FUNCTION_BLOCK Test_F_Equals EXTENDS TUnitTestBase
VAR
END_VAR

Assertion.AssertEquals_BOOL(
    Expected:= TRUE, 
    Actual:= F_Equals(1.000_005,1.000_004,0.000_002), 
    VariableName:= 'F_Equals');
    
Assertion.AssertEquals_BOOL(
    Expected:= FALSE, 
    Actual:= F_Equals(1.000_005,1.000_003,0.000_001), 
    VariableName:= 'F_Equals');
    
TestFinished();

END_FUNCTION_BLOCK

(* stored: Version 1.1.0.1, ProductVersion 3.1.4024.4
   POU Test_F_Equals: Id {c9fce891-e38b-43a8-928c-313315d741ad}, SpecialFunc None *)
